// TIA Portal V18 export
FUNCTION_BLOCK "UVLamp"   // FB19, LAD
TITLE = Description
{ S7_Optimized_Access := 'TRUE' }
VERSION : 0.1
// How to control and set the UV lamp:
// To control the lamp the machine needs to be started, all door closed and "LampFaultSignal" checked. After setting the setpoint 0-100 "LampSetpointInput" and enabling "LampEnable", the UV will work.
// 
// SafetyLimitSet - can be used to modify output range 
// 
// E-STOP - always check!
// stored: AutoNumber true, IsIECCheckEnabled false, IsRetainMemResEnabled false, MemoryReserve 100, SetENOAutomatically false, UDAEnableTagReadback false
   VAR_INPUT
      Emergency : Bool;
      MachineStart : Bool;
      LampEnable : Bool;   // Device ready do use
      LampMode : Int;   // 0 by default
      LampSetpointInput : Real;   // Intensity %
      LampMaintenance : Int;   // N/A
      LampFaultSignal : Bool;   // Signal from the UV lamp
      DoorSensor : Bool;   // Connect direct
      XPosition : DInt;
      YPosition : DInt;
      WorkingRegionXstart : DInt;   // To be updated and connected to the UV lamp preferences in the MachineDB
      WorkingRegionXend : DInt := 500000;   // To be updated and connected to the UV lamp preferences in the MachineDB
      WorkingRegionYstart : DInt;   // To be updated and connected to the UV lamp preferences in the MachineDB
      WorkingRegionYend : DInt := 1500000;   // To be updated and connected to the UV lamp preferences in the MachineDB
      DevelopmentMode : Bool;
      FirstTurnOn : Bool;
   END_VAR
   VAR_OUTPUT
      LampEnabled : Bool;
      LampWorking : Bool;
      LampOutONOFF : Bool;
      LampDimming : UInt;
      LampIntensity : Real;   // Volts
      LampError : Bool;
      LampStatus : Int;   // N/A
   END_VAR
   VAR_IN_OUT
      LampInONOFF : Bool;   // Device use state
   END_VAR
   VAR
      InternalWorkingPermission : Bool;
      SetpointMax : UInt := 27648;   // 0 - 0V; 27648 - 10V;
      SetpointLimit : UInt := 27648;
      SetpointConversion : Real;
      SetpointOutput : UInt;
      SafetyLimitConversion : Real;
      IntensityConversion : Real;
   END_VAR
   VAR_TEMP
      WorkingRegionOK : Bool;
   END_VAR
   VAR CONSTANT
      SafetyLimitSet : Real := 60.0;   // 0-100%
   END_VAR
BEGIN

REGION Network 1: Working Region Check
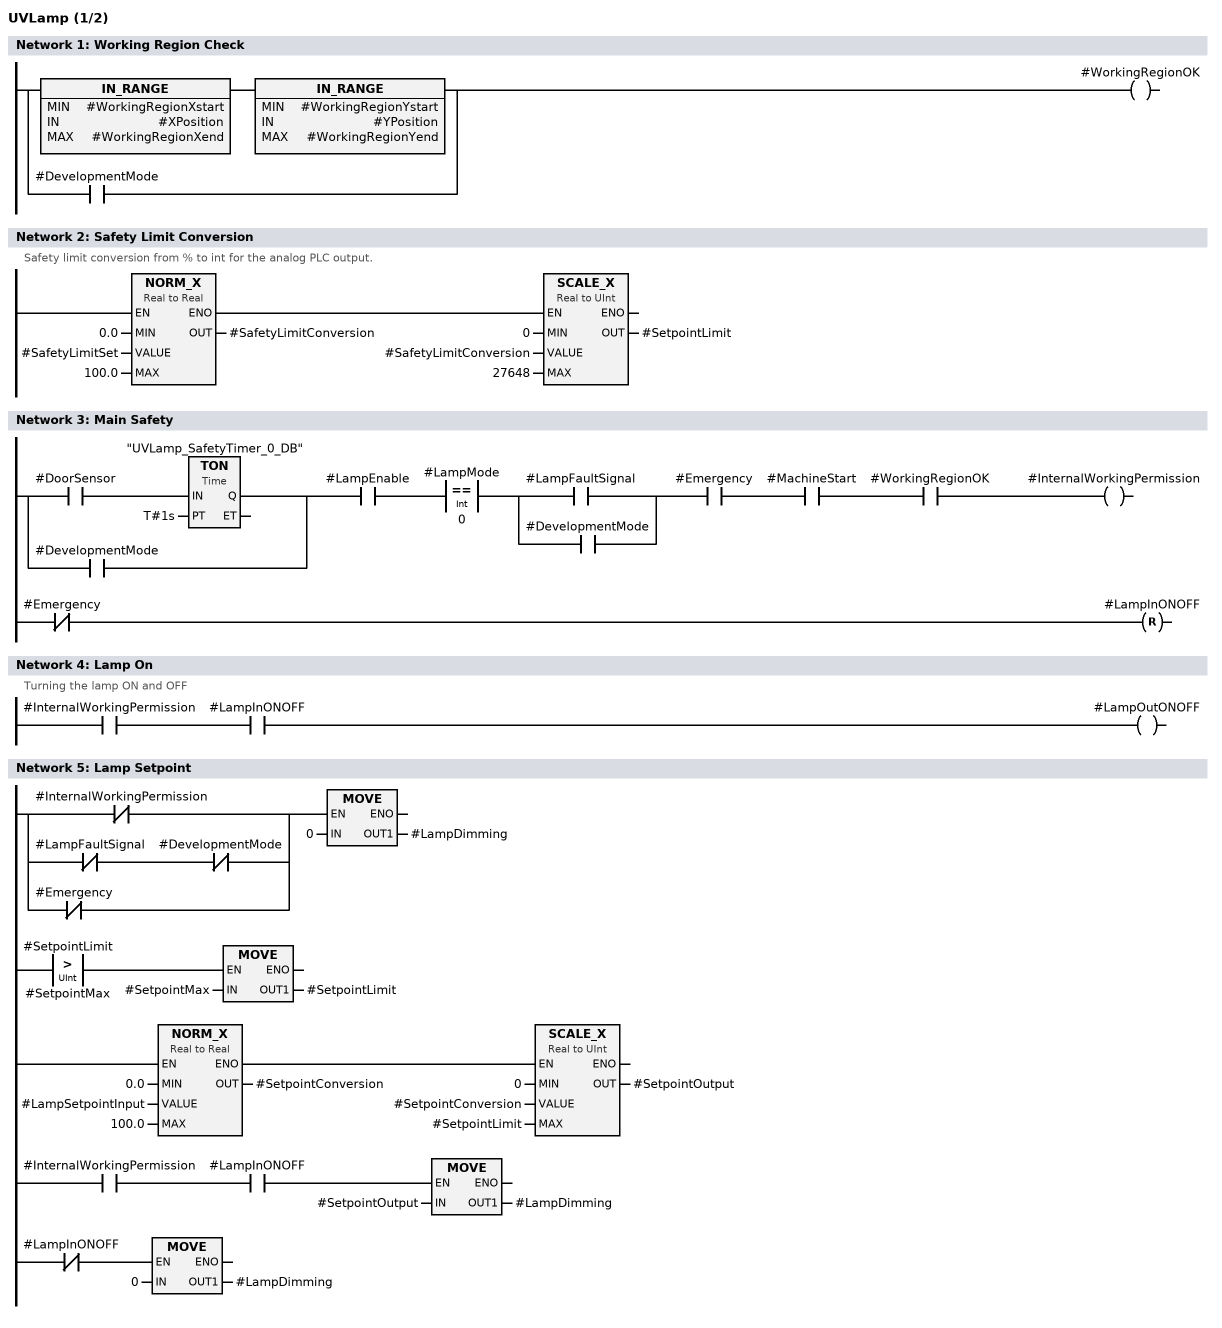
   RUNG wire#powerrail
      { S7_Templates := "SrcType := DInt" } InRange(min := #WorkingRegionXstart, in := #XPosition, max := #WorkingRegionXend)
      { S7_Templates := "SrcType := DInt" } InRange(min := #WorkingRegionYstart, in := #YPosition, max := #WorkingRegionYend)
      wire#w1
      Coil( #WorkingRegionOK )
   END_RUNG
   RUNG wire#powerrail
      Contact( #DevelopmentMode )
   END_RUNG wire#w1
   // the same network as SCL:
   #WorkingRegionOK := ((#WorkingRegionXstart <= #XPosition) AND (#XPosition <= #WorkingRegionXend) AND (#WorkingRegionYstart <= #YPosition) AND (#YPosition <= #WorkingRegionYend)) OR #DevelopmentMode;
END_REGION

REGION Network 2: Safety Limit Conversion
   // Safety limit conversion from % to int for the analog PLC output.
   RUNG wire#powerrail
      { S7_Templates := "[SrcType := Real, DestType := Real]" } Normalize(min := 0.0, value := #SafetyLimitSet, max := 100.0, out => #SafetyLimitConversion)
      { S7_Templates := "[SrcType := Real, DestType := UInt]" } Scale(min := 0, value := #SafetyLimitConversion, max := 27648, out => #SetpointLimit)
   END_RUNG
   // the same network as SCL:
   #SafetyLimitConversion := NORM_X(MIN := 0.0, VALUE := #SafetyLimitSet, MAX := 100.0);
   #SetpointLimit := SCALE_X(MIN := 0, VALUE := #SafetyLimitConversion, MAX := 27648);
END_REGION

REGION Network 3: Main Safety
   RUNG wire#powerrail
      Contact( #DoorSensor )
      { S7_Templates := "time_type := Time" } "UVLamp_SafetyTimer_0_DB".TON(pt := T#1s, et =>)
      wire#w1
      Contact( #LampEnable )
      { S7_Templates := "SrcType := Int" } EQ_Contact(in1 := #LampMode, in2 := 0)
      wire#w2
      Contact( #LampFaultSignal )
      wire#w3
      Contact( #Emergency )
      Contact( #MachineStart )
      Contact( #WorkingRegionOK )
      Coil( #InternalWorkingPermission )
   END_RUNG
   RUNG wire#powerrail
      Contact( #DevelopmentMode )
   END_RUNG wire#w1
   RUNG wire#w2
      Contact( #DevelopmentMode )
   END_RUNG wire#w3
   RUNG wire#powerrail
      I_Contact( #Emergency )
      R_Coil( #LampInONOFF )
   END_RUNG
   // the same network as SCL:
   "UVLamp_SafetyTimer_0_DB".TON(IN := #DoorSensor, PT := T#1s);
   #InternalWorkingPermission := ("UVLamp_SafetyTimer_0_DB".Q OR #DevelopmentMode) AND #LampEnable AND (#LampMode = 0) AND (#LampFaultSignal OR #DevelopmentMode) AND #Emergency AND #MachineStart AND #WorkingRegionOK;
   IF NOT #Emergency THEN #LampInONOFF := FALSE; END_IF;
END_REGION

REGION Network 4: Lamp On
   // Turning the lamp ON and OFF
   RUNG wire#powerrail
      Contact( #InternalWorkingPermission )
      Contact( #LampInONOFF )
      Coil( #LampOutONOFF )
   END_RUNG
   // the same network as SCL:
   #LampOutONOFF := #InternalWorkingPermission AND #LampInONOFF;
END_REGION

REGION Network 5: Lamp Setpoint
   RUNG wire#powerrail
      I_Contact( #InternalWorkingPermission )
      wire#w1
      Move(in := 0, out1 => #LampDimming)
   END_RUNG
   RUNG wire#powerrail
      I_Contact( #LampFaultSignal )
      I_Contact( #DevelopmentMode )
   END_RUNG wire#w1
   RUNG wire#powerrail
      I_Contact( #Emergency )
   END_RUNG wire#w1
   RUNG wire#powerrail
      { S7_Templates := "SrcType := UInt" } GT_Contact(in1 := #SetpointLimit, in2 := #SetpointMax)
      Move(in := #SetpointMax, out1 => #SetpointLimit)
   END_RUNG
   RUNG wire#powerrail
      { S7_Templates := "[SrcType := Real, DestType := Real]" } Normalize(min := 0.0, value := #LampSetpointInput, max := 100.0, out => #SetpointConversion)
      { S7_Templates := "[SrcType := Real, DestType := UInt]" } Scale(min := 0, value := #SetpointConversion, max := #SetpointLimit, out => #SetpointOutput)
   END_RUNG
   RUNG wire#powerrail
      Contact( #InternalWorkingPermission )
      Contact( #LampInONOFF )
      Move(in := #SetpointOutput, out1 => #LampDimming)
   END_RUNG
   RUNG wire#powerrail
      I_Contact( #LampInONOFF )
      Move(in := 0, out1 => #LampDimming)
   END_RUNG
   // the same network as SCL:
   IF NOT #InternalWorkingPermission OR (NOT #LampFaultSignal AND NOT #DevelopmentMode) OR NOT #Emergency THEN
       #LampDimming := 0;
   END_IF;
   IF #SetpointLimit > #SetpointMax THEN #SetpointLimit := #SetpointMax; END_IF;
   #SetpointConversion := NORM_X(MIN := 0.0, VALUE := #LampSetpointInput, MAX := 100.0);
   #SetpointOutput := SCALE_X(MIN := 0, VALUE := #SetpointConversion, MAX := #SetpointLimit);
   IF #InternalWorkingPermission AND #LampInONOFF THEN #LampDimming := #SetpointOutput; END_IF;
   IF NOT #LampInONOFF THEN #LampDimming := 0; END_IF;
END_REGION

REGION Network 6: Intensity Monitoring Conversion
   // Conversion of the intensity.
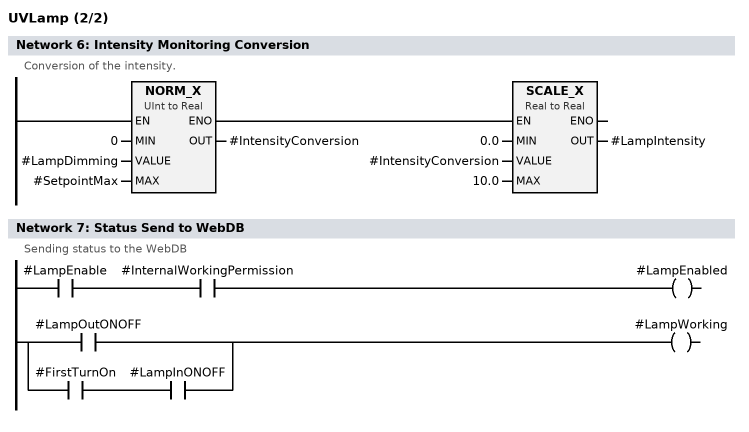
   RUNG wire#powerrail
      { S7_Templates := "[SrcType := UInt, DestType := Real]" } Normalize(min := 0, value := #LampDimming, max := #SetpointMax, out => #IntensityConversion)
      { S7_Templates := "[SrcType := Real, DestType := Real]" } Scale(min := 0.0, value := #IntensityConversion, max := 10.0, out => #LampIntensity)
   END_RUNG
   // the same network as SCL:
   #IntensityConversion := NORM_X(MIN := 0, VALUE := #LampDimming, MAX := #SetpointMax);
   #LampIntensity := SCALE_X(MIN := 0.0, VALUE := #IntensityConversion, MAX := 10.0);
END_REGION

REGION Network 7: Status Send to WebDB
   // Sending status to the WebDB
   RUNG wire#powerrail
      Contact( #LampEnable )
      Contact( #InternalWorkingPermission )
      Coil( #LampEnabled )
   END_RUNG
   RUNG wire#powerrail
      Contact( #LampOutONOFF )
      wire#w1
      Coil( #LampWorking )
   END_RUNG
   RUNG wire#powerrail
      Contact( #FirstTurnOn )
      Contact( #LampInONOFF )
   END_RUNG wire#w1
   // the same network as SCL:
   #LampEnabled := #LampEnable AND #InternalWorkingPermission;
   #LampWorking := #LampOutONOFF OR (#FirstTurnOn AND #LampInONOFF);
END_REGION
END_FUNCTION_BLOCK
